FUNCTION_BLOCK LiftSensor
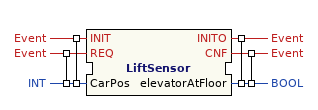
  EVENT_INPUT
    INIT WITH CarPos;
    REQ WITH CarPos;
  END_EVENT
  EVENT_OUTPUT
    INITO WITH elevatorAtFloor;
    CNF WITH elevatorAtFloor;
  END_EVENT
  VAR_INPUT
    CarPos : INT;
  END_VAR
  VAR_OUTPUT
    elevatorAtFloor : BOOL;
  END_VAR
  VAR
    prevPos : INT;
  END_VAR
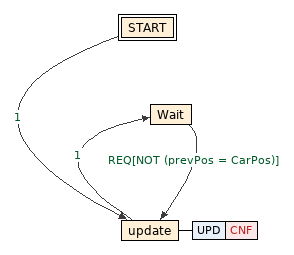
  EC_STATES
    START;
    update : UPD -> CNF;
    Wait;
  END_STATES
  EC_TRANSITIONS
    Wait TO update := REQ[NOT (prevPos = CarPos)];
    update TO Wait := 1;
    START TO update := 1;
  END_TRANSITIONS
  ALGORITHM initialize IN ST:
position := CarPos;&#38;#10;
  END_ALGORITHM
  ALGORITHM UPD IN ST:
elevatorAtFloor[0] := CarPos = 1;&#38;#10;elevatorAtFloor[1] := CarPos = 3;&#38;#10;elevatorAtFloor[2] := CarPos = 5;&#38;#10;elevatorAtFloor[3] := CarPos = 7;&#38;#10;elevatorAtFloor[4] := CarPos = 9;&#38;#10;prevPos := CarPos;&#38;#10;
  END_ALGORITHM
END_FUNCTION_BLOCK
